(* CoDeSys 2.3.9.45 project: FUP.pro *)
(* Libraries: Standard.lib 2.12.10 14:48:34, SYSLIBCALLBACK.LIB 2.12.10 14:48:32 *)

(* PLC configuration (modules and I/O channels)
K-Bus [K_Bus] node 0, in %IB0 out %QB0
Fieldbus variables [FB_VARS] node 1, in %IB0 out %QB0
Flag variables [FLAG_VARS] node 2, in %IB0 out %QB0
Modbus-Master [MB_MASTER] node 3, in %IB0 out %QB0
*)

(* POU PLC_PRG, FBD *)
PROGRAM PLC_PRG
VAR
	K1: BOOL;
	DELAY: TOF;
	TDELAY: TIME;
END_VAR
VAR_INPUT
	S8: BOOL;
	S1: BOOL;
END_VAR
VAR_OUTPUT
	K2: BOOL;
	L: BOOL;
END_VAR
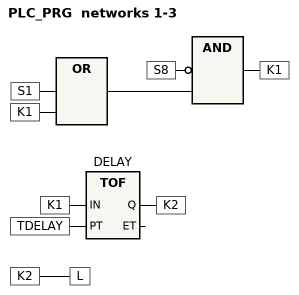
_FBD_ (* Function Block Diagram *)
NETWORK 1
	AND(NOT S8, OR(S1, K1)) => K1
NETWORK 2
	DELAY:TOF(IN: K1, PT: TDELAY) => K2
NETWORK 3
	K2 => L
_END_FBD_
(* the same logic as Structured Text *)
(* Network 1 *)
K1 := NOT S8 AND (S1 OR K1);
(* Network 2 *)
DELAY(IN := K1, PT := TDELAY);
K2 := DELAY.Q;
(* Network 3 *)
L := K2;
END_PROGRAM
